KUKA KRL data list: TurnOffRSI.dat

&ACCESS RV1
DEFDAT  TurnOffRSI PUBLIC

ENDDAT
